SUBAPPLICATION IN_UP (* Subapplication Type *)
  (* Standard: 61499-2 *)
  (* Version 1.0, 2023-02-06, franz *)
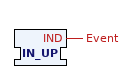
  EVENT_OUTPUT
    IND;
  END_EVENT
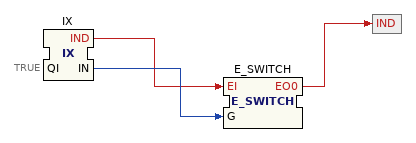
  FBS
    E_SWITCH : E_SWITCH;
    IX : IX(QI := TRUE);
  END_FBS
  EVENT_CONNECTIONS
    IX.IND TO E_SWITCH.EI;
    E_SWITCH.EO0 TO IND;
  END_CONNECTIONS
  DATA_CONNECTIONS
    IX.IN TO E_SWITCH.G;
  END_CONNECTIONS
END_SUBAPPLICATION
